TYPE ST_BA_BuildingSunblind :
STRUCT
	bGlobalThAuto_Release			: BOOL;
	bGlobalTwiLgtAuto_Release		: BOOL;
	nSunPrtc_PositionInterval		: UDINT;
	bIce							: BOOL;
	bGlobalResetManMode				: BOOL;	
END_STRUCT
END_TYPE

(* stored: Version 1.1.0.1, ProductVersion 3.1.4024.6
   DUT ST_BA_BuildingSunblind: Id {6ae73158-5d27-4399-8399-9948e4995717} *)
